FUNCTION_BLOCK FB_SequenceHelper
VAR_INPUT
	InHome		: BOOL; // in home helper status flag
	Busy		: BOOL; // busy helper status flag
	EnableStep	: BOOL; // enable step mode
END_VAR
VAR_OUTPUT
	Init,				// step init flag
	SeqRun		: BOOL; // sequence run flag 
	StepTime,			// step time
	SeqTime		: TIME;	// sequence time
END_VAR
VAR
	nStep,
	nStepMirror	: UINT;
	tonStep,
	tonSequence	: TON;
END_VAR

Init := nStepMirror <> Step;
tonStep(IN := nStepMirror = Step, PT := T#49D17H2M47S295MS);
StepTime := tonStep.ET;
tonSequence(IN := SeqRun, PT := T#49D17H2M47S295MS);
SeqTime := tonSequence.ET;
nStepMirror := Step;

METHOD PUBLIC Reset : REFERENCE TO FB_SequenceHelper
VAR_INPUT
	value : UINT := 0;
END_VAR
Reset REF= THIS^;
Step := value;
END_METHOD

METHOD PUBLIC SetStep : REFERENCE TO FB_SequenceHelper
VAR_INPUT
	value : UINT;
END_VAR
SetStep REF= THIS^;

IF EnableStep THEN
	Step := value;	
END_IF
END_METHOD

METHOD PUBLIC StartSequence : REFERENCE TO FB_SequenceHelper
VAR_INPUT
END_VAR
StartSequence REF= THIS^;
tonSequence(IN := FALSE);
SeqRun := TRUE;
END_METHOD

{attribute 'monitoring' := 'call'}
PROPERTY PUBLIC Step : UINT
GET
Step := nStep;
END_GET
SET
nStep := Step;
END_SET
END_PROPERTY

METHOD PUBLIC StopSequence : REFERENCE TO FB_SequenceHelper
VAR_INPUT
END_VAR
StopSequence REF= THIS^;
SeqRun := FALSE;
END_METHOD

END_FUNCTION_BLOCK

(* stored: Version 1.1.0.1
   POU FB_SequenceHelper: Id {ff57f4bf-8abe-4821-bdfd-ba3b55c414cf}, SpecialFunc None
   Method Reset: Id {71553e8b-85b1-4f76-8283-c6ab25b16daf}
   Method SetStep: Id {0f5adac3-0315-4816-8dc8-e25505104b69}
   Method StartSequence: Id {5ddb84e8-825b-4e8e-b146-56fe4081fc8e}
   Property Step: Id {0a02b69f-40d2-4b8c-9ea0-cdae45986433}
   Get Get: Id {de97d576-81c8-4f8d-9462-73c28c05342c}
   Set Set: Id {90fb912f-9db6-4dec-bd2f-a882a9e3dbe8}
   Method StopSequence: Id {9e2dbdc3-8d4c-4d6a-9aeb-116371519af7} *)
